/// Zeugwerk Application
PROGRAM ZModuleProgram
VAR_INPUT
{region "ZModuleProgram : Utility"}
  App : ZApp(displayName:='Zeugwerk-Application Template', com:=ZGlobal.Com.App);
  Datetime : ZAux.DateTimeUM;
  {attribute 'ZId' := ''}
{endregion}
{region "ZModuleProgram : Logging"}
  Alarming : ZApplication.Alarming(App, datetime := Datetime, com := ZGlobal.Com.Alarming);
  LoggerHmi : ZApplication.Messaging(App, datetime := Datetime, com := ZGlobal.Com.Messages);
  LoggerFile : ZAux.LoggerFile7FF(App, datetime := Datetime, filePath:='C:\Zeugwerk\logs\messages.log', target:='');
  Logger : ZAux.Logging;
  {attribute 'ZId' := ''}
{endregion}  
{attribute '__ZwPlcApplicationModuleProgramDeclaration__'} // Do not remove this attribute! It is used for code generation.
{region "XyTable"}
{undefine RunInSeparateProgram}
{IF NOT (defined (XyTable_disabled)) AND NOT (defined (RunInSeparateProgram))}
  XyTable : XyTableUnit(name := 'XyTable', // name of the unit (for logging)
					  parent := App, // caller of the Unit's cyclic method. If the Unit runs in its own context use 0
						configdata := ZGlobal.Data.Config.XyTable,
						machinedata := ZGlobal.Data.Machine.XyTable,
						calibrationdata := ZGlobal.Data.Calibration.XyTable,
						com := ZGlobal.Com.Unit.XyTable);
  {attribute 'section' := '__ZwPlcUnitProgramDeclaration__'}
  {attribute 'ZId' := '934662f7-81a9-4247-b804-76d465c7ec61'}
{END_IF}
{endregion}
{attribute '__ZwPlcUnitProgramDeclaration__'} // Do not remove this attribute! It is used for code generation.
END_VAR

{region "ZModuleProgram : Utility"}
  Datetime.Cyclic();
  App.Cyclic();
  {attribute 'ZId' := ''}
{endregion}
{attribute '__ZwPlcApplicationModuleProgramImplementation__'} // Do not remove this attribute! It is used for code generation.

END_PROGRAM

(* stored: Version 1.1.0.1
   POU ZModuleProgram: Id {a120f957-5953-492b-ac4f-29b84ddfacdc}, SpecialFunc None *)
